TYPE s_DataSample :
STRUCT
	DataSet :  ARRAY[0..500] OF s_DataSampleCav;
	SetQty	:  s_DataSampleCav_setQty;
END_STRUCT
END_TYPE

(* stored: Version 1.1.0.1, ProductVersion 3.1.4024.11
   DUT s_DataSample: Id {4f0beae9-e8e0-44be-a4d3-1f11dcb4f63b} *)
